// TwinCAT 3 PLC project Main
// ProgramVersion: 3.1.4026.10
// libraries:
//   Tc2_EtherCAT, * (Beckhoff Automation GmbH)
//   Tc2_IoFunctions, * (Beckhoff Automation GmbH)
//   Tc2_Math, * (Beckhoff Automation GmbH)
//   Tc2_MC2, * (Beckhoff Automation GmbH)
//   Tc2_NC, * (Beckhoff Automation GmbH)
//   Tc2_Standard, * (Beckhoff Automation GmbH)
//   Tc2_System, * (Beckhoff Automation GmbH)
//   Tc2_Utilities, * (Beckhoff Automation GmbH)
//   Tc3_EventLogger, * (Beckhoff Automation GmbH)
//   Tc3_McCollisionAvoidance, * (Beckhoff Automation GmbH)
//   Tc3_McCoordinatedMotion, * (Beckhoff Automation GmbH)
//   Tc3_Module, * (Beckhoff Automation GmbH)
//   Tc3_XTS_Utility, * (Beckhoff Automation GmbH)
// project tree:
//   DUTs/delete/ MainCommands_typ.TcDUT, MainStateMachine_enum.TcDUT (not stored), MainState_enum.TcDUT, MediatorGroupStatus.TcDUT (not stored), MotionParameters_typ.TcDUT (not stored), MoverCommandType_enum.TcDUT (not stored), MoverState_enum.TcDUT (not stored), PositionTriggerStats_typ.TcDUT (not stored), StationStats_typ.TcDUT (not stored), TrackCyclicState.TcDUT (not stored), TrackInfo.TcDUT (not stored), TrackState.TcDUT (not stored), UserStationsMonitor.TcDUT (not stored)
//   DUTs/ M1Detection.TcDUT (not stored), MoverControlFlags.TcDUT, MoverSequence.TcDUT, StationSequence.TcDUT (not stored), XTSSequence.TcTLEO
//   / GlobalTextList.TcGTLO (not stored), PlcTask.TcTTO
//   GVLs/ GVL.TcGVL, HMI.TcGVL, IOGVL.TcGVL, SafetyGVL.TcGVL
//   ITFs/ iMoverList.TcIO (not stored), iMover.TcIO, iTrack.TcIO (not stored)
//   POUs/ Main.TcPOU
//   POUs/XTS/ Mover.TcPOU, Station.TcPOU, Zone.TcPOU

CONFIGURATION Main
    RESOURCE PLC ON TwinCAT3
        TASK PlcTask(INTERVAL := T#1ms, PRIORITY := 6);
        PROGRAM Main WITH PlcTask : Main;
    END_RESOURCE
END_CONFIGURATION

// ---- DUTs/delete/MainCommands_typ.TcDUT
TYPE MainCommands_typ :
    STRUCT

        Enable  : BOOL; // Enables Movers & Collision Avoidance, activates M1 Detection
        Start   : BOOL; // Issues initial command, starts motion
        Stop    : BOOL; // Stops movers, deregisters movers from all objectives	
        Disable : BOOL; // Disables Movers, Ungroups Movers

    END_STRUCT
END_TYPE

// ---- DUTs/delete/MainState_enum.TcDUT
{attribute 'strict'}
{attribute 'to_string'}
TYPE MainState_enum : (
        MS_DISABLED					:= 0,
		MS_INITIALIZING_XPU			:= 5,
        MS_INITIALIZING_MOVERS		:= 10,
		MS_ONESHOT_ENABLE			:= 20,
        MS_ENABLING_MOVERS			:= 30,
        MS_INITIALIZING_OBJECTIVES	:= 40,
		MS_INITIALIZE_TRACKS		:= 44,
		MS_ACTIVATE_TRACKS			:= 45,
		MS_WAIT_FOR_TRACKS			:= 46,
        MS_ENABLED					:= 50,
        MS_RUN						:= 60,
		MS_ONESHOT_STOP				:= 70,
        MS_STOPPING					:= 80,
        MS_STOPPED					:= 90,
		MS_ONESHOT_DISABLE			:= 100,
        MS_DISABLING				:= 110,
        MS_ERROR					:= 120,
        MS_DEBUG					:= 1000
    );
END_TYPE

// ---- DUTs/MoverControlFlags.TcDUT
TYPE MoverControlFlags :
STRUCT

	loadTray_Busy		: BOOL;			// To the machine to check Sensor
	loadTray_Complete	: BOOL;			// From Sensor is TRUE
	loadArea1_Busy		: BOOL;			// TO Robot 1 to start working
	loadArea1_Complete	: BOOL;			// FROM Robot 1 that placing parts has completed
	loadArea2_Busy		: BOOL;			// TO Robot 2 to start working
	loadArea2_Complete	: BOOL;			// FROM Robot 1 that placing parts has completed
	loadArea3_Busy		: BOOL;			// TO Robot 3 to start working
	loadArea3_Complete	: BOOL;			// FROM Robot 1 that placing parts has completed
	loadArea4_Busy		: BOOL;			// TO Robot 4 to start working
	loadArea4_Complete	: BOOL;			// From Robot 1 that placing parts has completed
	unloadTray_Busy		: BOOL;			// To Robot 5 to start working
	unloadTray_Complete	: BOOL;			// From Robot 5. Tray is unloaded



END_STRUCT
END_TYPE

// ---- DUTs/MoverSequence.TcDUT
{attribute 'qualified_only'}
{attribute 'strict'}
TYPE MoverSequence :
(
	Off,
	Idle,
	MovingToStart,
	AtStart,
	MovingToStation,
	AtStation,
	MovingToQueue,
	AtQueue,
	Error,
	Stop,
	Stopping,
	RemoveAxes,
	RemovingAxes,
	Pausing,
	Paused,
	Disabling,
	Disabled,
	Reset,
	Resetting,
	Waiting	
);
END_TYPE

// ---- DUTs/XTSSequence.TcTLEO
{attribute 'qualified_only'}
{attribute 'strict'}
TYPE XTSSequence :
(
	Off,
	EnableMovers,
	EnableGroup,
	AddAxes,
	RemoveAxes,
	RemovedAxes,
	DisableMovers,
	Disabled,
	Start,
	Run,
	Stop,
	Stopping,
	Paused,
	Standby,
	Error,
	Waiting
);
END_TYPE

// ---- GVLs/GVL.TcGVL
{attribute 'qualified_only'}
VAR_GLOBAL CONSTANT

    pXtsProcessingUnit : OTCID	:=	01010090;	 

	TRACK_LENGTH 				: LREAL := 7000; // This should be set to the exact length [mm] of the track system
	NUM_MOVERS   				: USINT := 20;   // This should be set to the exact number of movers on the system
	
	// The following should be set to a value **equal to or greater than** the number of objectives needed
	NUM_POSITIONTRIGGERS		: USINT := 10;	// Position Triggers
	NUM_STATIONS				: USINT := 8;	// Stations
	NUM_ZONES					: USINT := 10;	// Zones

	// Station constants
	startStation				: USINT	:= 1;		// set this number to the index of the station all movers should start from
	stationTolerance			: LREAL	:= 0.5;		// set to number of millimeters tolerance for mover at station
	zeroSpeed					: LREAL	:= 10.0;		// tolerance for definition of not moving

END_VAR
VAR_GLOBAL
	Mover			: ARRAY[1..GVL.NUM_MOVERS] OF Mover;
	Station			: ARRAY[1..GVL.NUM_STATIONS] OF station;
	Zone			: ARRAY[1..GVL.NUM_ZONES] OF zone;
	newCallTime: LREAL;
	
	//-------------ADDED BY NIJAZ-------------
	dsMoverControlFlags		:	MoverControlFlags;
	
END_VAR

// ---- GVLs/HMI.TcGVL
{attribute 'qualified_only'}
VAR_GLOBAL
	Start					: BOOL;
	E_Stop					: BOOL;
	Stop					: BOOL;
	Resume					: BOOL;
	ResetXTS_Error			: BOOL;
	bzone0Stop				: BOOL;
	SafeToUnlock			: BOOL;
	dsMoverControlFlags		: MoverControlFlags;
	ShuttleMover			: BOOL;
	
	
	//Linked to SAFETY Alias
	LockDoors		AT %Q*	: BOOL;		
	
END_VAR

// ---- GVLs/IOGVL.TcGVL
{attribute 'qualified_only'}
VAR_GLOBAL
	
//INPUTS
iTrayDetectSensor	AT %I*	:	BOOL;
iDoor1Opened		AT %I*	:	BOOL;		
iDoor2Opened		AT %I*	:	BOOL;
iDoor3Opened		AT %I*	:	BOOL;
iDoor4Opened		AT %I*	:	BOOL;
iMainAirPressure 	AT %I*	:	BOOL;

//------XTS Power Monitor Breakers	
//- EL1809 Mod1
iCircuitBreaker24VDC			AT %I*	:	BOOL;
iCircuitBreakerSafety			AT %I*	:	BOOL;
iXTS_Module1					AT %I*	:	BOOL;
iXTS_Module2					AT %I*	:	BOOL;
iXTS_Module3					AT %I*	:	BOOL;
iXTS_Module4					AT %I*	:	BOOL;
iXTS_Module5					AT %I*	:	BOOL;
iXTS_Module6					AT %I*	:	BOOL;
iLubricationOn					AT %I*	:	BOOL;
//- EL1809 Mod2
iPowerSupply48VDC1				AT %I*	:	BOOL;
iPowerSupply48VDC2				AT %I*	:	BOOL;
iPowerSupply48VDC3				AT %I*	:	BOOL;
iLubricationLevelOK				AT %I*	:	BOOL;
iLubricationDone				AT %I*	:	BOOL;
iCircuitBreaker48VDC1			AT %I*	:	BOOL;
iCircuitBreaker48VDC2			AT %I*	:	BOOL;
iCircuitBreaker48VDC3			AT %I*	:	BOOL;
iCircuitBreakerXTSModule1		AT %I*	:	BOOL;
iCircuitBreakerXTSModule2		AT %I*	:	BOOL;
iCircuitBreakerXTSModule3		AT %I*	:	BOOL;
iCircuitBreakerXTSModule4		AT %I*	:	BOOL;
iCircuitBreakerXTSModule5		AT %I*	:	BOOL;
iCircuitBreakerXTSModule6		AT %I*	:	BOOL;
iBrakeResistorON				AT %I*	:	BOOL;

//-----------------------------------------------------------------------------------------------------------------------------------
//OUTPUTS
oBacklight1			AT %Q*	:	BOOL;
oBacklight2			AT %Q*	:	BOOL;
oBacklight3			AT %Q*	:	BOOL;
oBacklight4			AT %Q*	:	BOOL;
oBacklight5			AT %Q*	:	BOOL;
oBacklight6			AT %Q*	:	BOOL;
oBacklight7			AT %Q*	:	BOOL;
oBacklight8			AT %Q*	:	BOOL;
oBacklight9			AT %Q*	:	BOOL;
oBacklight10		AT %Q*	:	BOOL;
oBacklight11		AT %Q*	:	BOOL;
oBacklight12		AT %Q*	:	BOOL;
oBacklight13		AT %Q*	:	BOOL;
oBacklight14		AT %Q*	:	BOOL;
oBacklight15		AT %Q*	:	BOOL;
oBacklight16		AT %Q*	:	BOOL;
oEStopLight			AT %Q*	:	BOOL;
oConveyor			AT %Q*	:	BOOL;
oLubeON				AT %Q*	:	BOOL;


END_VAR

// ---- GVLs/SafetyGVL.TcGVL
{attribute 'qualified_only'}
VAR_GLOBAL
	
//OUTPUTS TO SAFETY GROUP
err_ack			AT %Q*	:	BOOL;
run				AT %Q*	:	BOOL := TRUE;
DoorsClosed 	AT %Q*	:	BOOL;
ResetCurtains	AT %Q*	:	BOOL;

//INPUTS FROM SAFETY GROUP
CurtainsOK		AT %I*	:	BOOL;
AllSafetyOK		AT %I*	:	BOOL;
EStopStatus		AT %I*	:	BOOL;

END_VAR

// ---- ITFs/iMover.TcIO
INTERFACE iMover

METHOD ActivateTrack : BOOL
VAR_INPUT
	Track	: REFERENCE TO Track;
END_VAR
END_METHOD

{attribute 'monitoring' := 'call'}
PROPERTY CurrentDestinationPosition : LREAL
GET
END_GET
END_PROPERTY

PROPERTY CurrentDestinationTrack : DINT
GET
END_GET
END_PROPERTY

{attribute 'monitoring' := 'call'}
PROPERTY CurrentMoveType : MoverCommandType_enum
GET
END_GET
END_PROPERTY

PROPERTY CurrentObjective : String
GET
END_GET
END_PROPERTY

PROPERTY CurrentTrack : POINTER TO Track
GET
END_GET
END_PROPERTY

METHOD Cyclic : iMover
VAR_IN_OUT
	GroupReference		: AXES_GROUP_REF;
END_VAR
END_METHOD

METHOD Disable : iMover
VAR_INPUT
END_VAR
END_METHOD

METHOD Enable : iMover
VAR_INPUT
END_VAR
END_METHOD

METHOD GroupStop : iMover
VAR_INPUT
END_VAR
END_METHOD

METHOD Halt : iMover
VAR_INPUT
END_VAR
END_METHOD

PROPERTY IsTrackReady : BOOL
GET
END_GET
END_PROPERTY

METHOD LogUserEvent : iMover
VAR_INPUT
	String1	: STRING;	// First content section of user-event message
	String2 : STRING;	// Second content section of user-event message
	String3 : STRING;	// Third content section of user-event message
END_VAR
END_METHOD

METHOD PUBLIC MoveToPosition : iMover
VAR_INPUT
	
	DestinationPosition		: LREAL;	// position on track for a shuttle to move towards

END_VAR
END_METHOD

METHOD MoveToStation : iMover
VAR_INPUT
	DestinationStation	: REFERENCE TO delete_Station;	
END_VAR
END_METHOD

METHOD MoveVelocity : iMover
VAR_INPUT
	DesiredVelocity : LREAL;		//The velocity to be commanded [mm/s]
END_VAR
END_METHOD

PROPERTY Payload : USINT
GET
END_GET
SET
END_SET
END_PROPERTY

METHOD ReissueCommand : iMover
VAR_INPUT
END_VAR
END_METHOD


METHOD SetAcceleration : iMover
VAR_INPUT
	Acceleration	: LREAL;
END_VAR
END_METHOD

METHOD SetDeceleration : iMover
VAR_INPUT
	Deceleration	: LREAL;
END_VAR
END_METHOD

METHOD SetDirection : iMover
VAR_INPUT
	Direction		: Tc3_Mc3Definitions.MC_Direction;
END_VAR
END_METHOD

METHOD SetGap : iMover
VAR_INPUT
	Gap	: LREAL;
END_VAR
END_METHOD

METHOD SetGapMode : iMover
VAR_INPUT
	Mode	: MC_GAP_CONTROL_MODE;
END_VAR
END_METHOD

METHOD SetJerk : iMover
VAR_INPUT
	Jerk		: LREAL;
END_VAR
END_METHOD

METHOD SetVelocity : iMover
VAR_INPUT
	Velocity		: LREAL;		// Updates Mover's internal velocity parameter. Takes effect immediately. [mm/s]
END_VAR
END_METHOD

METHOD SyncToAxis : iMover
VAR_INPUT
	
	MasterAxis		: REFERENCE TO AXIS_REF;
	MasterSyncPos	: LREAL;	// Master sync position (nonmodulo), where the input axis will be located when first synchronized
	SlaveSyncPos	: LREAL;	// Mover sync position, where the mover will be located when first synchronized
	SyncStrategy	: MC_SYNC_STRATEGY;	// Direction input
	
END_VAR
END_METHOD

METHOD SyncToMover : iMover
VAR_INPUT

	MasterMover		: REFERENCE TO delete_Mover;	// Synchronization master mover, whose position to follow. Further motion commands break the pairing
	Gap				: LREAL;				// Gap distance to lead mover. Positive values indicate following, negative values indicate leading

END_VAR
END_METHOD

END_INTERFACE

// ---- POUs/Main.TcPOU
PROGRAM Main
VAR
	PowerOn					: BOOL	:= TRUE;	// initialize on, turn false on second scan
	FirstRun				: BOOL := TRUE;		// initialize on, turn false when system has reached starting postion 
	i						: UINT;								// loop index variable
	Step					: XTSSequence;						// primary sequencer
	stCaGroupRef			: AXES_GROUP_REF;
	fbEnableGroup			: MC_GroupEnable;
	fbAddAxis				: ARRAY[1..GVL.NUM_MOVERS] OF MC_AddAxisToGroup;
	fbRemoveAxisFromGroup	: ARRAY[1..GVL.NUM_MOVERS] OF MC_RemoveAxisFromGroup;
	nAtStart				: UINT;
	nToStart				: UINT;
	allMoversHalted			: BOOL;	
	MoversReady				: BOOL;
	Started					: BOOL;		
	Resumed					: BOOL;
	bLightCurtainExited		: R_TRIG;
	bLightCurtainEntered	: F_TRIG;
	bEstopPressed			: F_TRIG;
	safeToOpenDoors			: BOOL;
	allMoversNotMoving		: BOOL;
	DelayMoversTimer		: TON;
	
	//Timers for generating a pulse
	PulseTON	: TON;
	PulseTOF	: TOF;
	OnDuration	: TIME := T#500MS;
	OFFDuration	: TIME := T#1000MS;
	bCycleBit	: BOOL;
	
	//M1 Detection
	fbReadM1DetectMode		: ADSREAD;
	fbReadM1DetectValid		: ADSREAD;
	fbReadM1DetectActive	: ADSREAD;
	fbWriteM1Detect			: ADSWRITE;
	fbDelayM1Timer			: TON;
	IsIdDetectionActive		: BOOL;			// M1 Detection currently underway
	Mover1Found				: BOOL;			// M1 Detection has completed
	Mover1Error				: BOOL;			// M1 Detection has Failed
	M1DetectStep			: M1Detection;	
	M1DetectAttemptCounter	: INT;
END_VAR

(* this program handles the main sequencer of this machine *)

// cyclic call to execute fb's for movers, stations, and zones
FOR i := 1 TO GVL.NUM_MOVERS DO
	GVL.Mover[i]();
	GVL.Mover[i].AxisReference.ReadStatus();
	fbRemoveAxisFromGroup[i](AxesGroup		:= stCaGroupRef);
	fbAddAxis[i](AxesGroup		:= stCaGroupRef,
				Axis			:= GVL.Mover[i].AxisReference);
	//Monitoring if all movers are in stopped motion state			
	IF GVL.Mover[i].AxisReference.Status.Moving THEN
		allMoversNotMoving	:= FALSE;
	ELSE
		allMoversNotMoving	:= TRUE;
	END_IF
	
END_FOR
FOR i := 1 TO GVL.NUM_STATIONS DO
	GVL.Station[i]();
END_FOR
FOR i := 1 TO gvl.NUM_ZONES DO
	GVL.Zone[i]();
END_FOR

IF HMI.ResetXTS_Error THEN
	FOR i := 1 TO GVL.NUM_MOVERS DO
		GVL.Mover[i].toReset := TRUE;
	END_FOR
	HMI.ResetXTS_Error := FALSE;
END_IF


// check for E-STOP
bEstopPressed(CLK:=SafetyGVL.EStopStatus);
IF bEstopPressed.Q OR HMI.E_Stop THEN
	Step			:= XTSSequence.Stop;
	HMI.E_Stop := FALSE;
END_IF

CASE Step OF

//-----------------------------------------------------------------------------------------------------------------------	
	XTSSequence.Off:
		IF SafetyGVL.EStopStatus AND IOGVL.iPowerSupply48VDC1 AND IOGVL.iPowerSupply48VDC2 AND IOGVL.iPowerSupply48VDC3 AND Mover1Found = FALSE THEN
			Initialize();
		END_IF
		// state waiting for HMI.Start
		IF HMI.Start AND Mover1Found THEN
			Step		:= XTSSequence.EnableMovers;
			Started 	:= TRUE;
			HMI.Start 	:= FALSE;
		END_IF

//-----------------------------------------------------------------------------------------------------------------------	
	XTSSequence.Paused:
		//state waiting for HMI.Start or HMI.Resume
		IF HMI.Start THEN
			Step		:= XTSSequence.EnableMovers;
			Started 	:= TRUE;
			HMI.Start 	:= FALSE;
		END_IF
	
		IF HMI.Resume THEN
			Step		:= XTSSequence.EnableMovers;
			Resumed 	:= TRUE;
			HMI.Resume 	:= FALSE;
			HMI.Stop  	:= FALSE;
		END_IF
	
//-----------------------------------------------------------------------------------------------------------------------	
	XTSSequence.Stop:
	
	FOR i := 1 TO GVL.NUM_MOVERS  DO
		GVL.Mover[i].toStop := TRUE;
	END_FOR
	
	Started 	:= FALSE;
	Resumed 	:= FALSE;
	Step		:= XTSSequence.Stopping;
		
//-----------------------------------------------------------------------------------------------------------------------	
	XTSSequence.Stopping:
		// Waiting for all to come to a full stop
		
	allMoversHalted		:= TRUE;
	
		FOR i := 1 TO GVL.NUM_MOVERS DO
			IF GVL.Mover[i].AxisReference.Status.Moving THEN
				allMoversHalted		:= FALSE;
			END_IF
		END_FOR
	
	IF allMoversHalted THEN
		Step		:= XTSSequence.RemoveAxes;
	END_IF
	
//-----------------------------------------------------------------------------------------------------------------------	
	XTSSequence.RemoveAxes:
		// remove all axes to collision avoidance group
		// loop through each mover axis and remove CA group
		FOR i:= 1 TO GVL.NUM_MOVERS DO
			fbRemoveAxisFromGroup[i].IdentInGroup := UDINT_TO_IDENTINGROUP(UINT_TO_UDINT(i));
			fbRemoveAxisFromGroup[i].Execute			:= TRUE;
		END_FOR
	
		IF stCaGroupRef.NcToPlc.CA.Common.GroupAxesCount = 0 THEN
			FOR i:= 1 TO GVL.NUM_MOVERS DO
				fbRemoveAxisFromGroup[i].IdentInGroup	:= UDINT_TO_IDENTINGROUP(UINT_TO_UDINT(i));
				fbRemoveAxisFromGroup[i].Execute			:= FALSE;
				MoversReady := FALSE;
		END_FOR
			Mover1Found := FALSE;
			Step := XTSSequence.DisableMovers;
		END_IF

//-----------------------------------------------------------------------------------------------------------------------	
	XTSSequence.DisableMovers:
	FOR i := 1 TO GVL.NUM_MOVERS  DO
		GVL.Mover[i].toDisable := TRUE;
	END_FOR
	
	Step := XTSSequence.Off;
		
//-----------------------------------------------------------------------------------------------------------------------			
	XTSSequence.EnableMovers:
		// enable all movers
		FOR i := 1 TO GVL.NUM_MOVERS DO
			IF NOT GVL.Mover[i].Enabled THEN
				GVL.Mover[i].Enable	:= TRUE;
			END_IF
		END_FOR
		
		// check for all enabled
		FOR i := 1 TO GVL.NUM_MOVERS DO
			IF NOT GVL.Mover[i].Enabled THEN
				// not enabled, leave for loop
				EXIT;
			END_IF
			// made it this far, all movers are enabled
			IF i = gvl.NUM_MOVERS THEN
				Step	:= XTSSequence.EnableGroup;
			END_IF
		END_FOR
		
//-----------------------------------------------------------------------------------------------------------------------		
	XTSSequence.EnableGroup:
	// enable CA group
	fbEnableGroup.Execute := TRUE;
	// verify group enabled successfully
	IF fbEnableGroup.Done = TRUE THEN
		fbEnableGroup.Execute := FALSE;
		Step := XTSSequence.AddAxes;
	END_IF
		
//-----------------------------------------------------------------------------------------------------------------------		
	XTSSequence.AddAxes:
		// add all axes to collision avoidance group
		// loop through each mover axis and add to CA group
	FOR i:= 1 TO GVL.NUM_MOVERS DO
		fbAddAxis[i].IdentInGroup := UDINT_TO_IDENTINGROUP(UINT_TO_UDINT(i));
		fbAddAxis[i].Execute := TRUE;
	END_FOR
	
	// verify all axes added
	IF stCaGroupRef.NcToPlc.CA.Common.GroupAxesCount = GVL.NUM_MOVERS THEN
		FOR i:= 1 TO GVL.NUM_MOVERS DO
			fbAddAxis[i].IdentInGroup := UDINT_TO_IDENTINGROUP(UINT_TO_UDINT(i));
			fbAddAxis[i].Execute := FALSE;
			Step	:= XTSSequence.StandBy;
		END_FOR
	END_IF
		
//-----------------------------------------------------------------------------------------------------------------------		
	XTSSequence.StandBy:
	IF Started THEN
		// first time code executes this far (after power on) move to a start position
		Started := FALSE;
		Step	:= XTSSequence.Start;
	ELSIF Resumed THEN
		// any other time code executes here, resume operation where movers left off
		Resumed := FALSE;
		Step	:= XTSSequence.Run;
	END_IF

//-----------------------------------------------------------------------------------------------------------------------		
	XTSSequence.Start:
		// request all movers proceed to starting station
IF HMI.bzone0Stop = FALSE THEN
	FOR i:= 1 TO GVL.NUM_MOVERS DO
		GVL.Mover[i].toStart	:= TRUE;
	END_FOR
	// verify one mover is at start, all others have commands and are at zero speed
	nAtStart	:= 0;
	nToStart	:= 0;
	FOR i:= 1 TO GVL.NUM_MOVERS DO
		IF GVL.Mover[i].Step = MoverSequence.AtStart THEN
			nAtStart	:= nAtStart + 1;
		ELSIF GVL.Mover[i].Step = MoverSequence.MovingToStart THEN
			nToStart	:= nToStart + 1;
		END_IF
	END_FOR
	IF nAtStart = 1 AND nToStart = GVL.NUM_MOVERS - 1 THEN
		Step	:= XTSSequence.Run;
	END_IF
END_IF	
//-----------------------------------------------------------------------------------------------------------------------	
	XTSSequence.Run:

IF HMI.Stop = FALSE THEN
	
	// LOAD TRAY STATION
	IF GVL.Station[1].Step = StationSequence.MoverPresent THEN
		HMI.dsMoverControlFlags.loadTray_Busy := TRUE;
		IF HMI.dsMoverControlFlags.loadTray_Complete THEN			//IF SENSOR IS TRUE PACKAGE IS PRESENT MOVER GOES TO NEXT STATION
			HMI.dsMoverControlFlags.loadTray_Complete := FALSE;
			GVL.Station[1].bMoveToNext := TRUE;
		END_IF
	ELSE
		HMI.dsMoverControlFlags.loadTray_Busy := FALSE;
	END_IF
	
	// INSPECT TRAY STATION
	IF GVL.Station[2].Step = StationSequence.MoverPresent THEN
		HMI.dsMoverControlFlags.inspectTray_Busy := TRUE;
		IF HMI.dsMoverControlFlags.inspectTray_Complate THEN			//IF SENSOR IS TRUE PACKAGE IS PRESENT MOVER GOES TO NEXT STATION
			HMI.dsMoverControlFlags.inspectTray_Complate := FALSE;
			GVL.Station[2].bMoveToNext := TRUE;
		END_IF
	ELSE
		HMI.dsMoverControlFlags.inspectTray_Busy := FALSE;
	END_IF
	
	// LOAD PARTS STATION 1
	IF GVL.Station[3].Step = StationSequence.MoverPresent THEN
		HMI.dsMoverControlFlags.loadArea1_Busy := TRUE;				//SIGNAL TO ROBOT 1 TO LOAD PARTS
		IF HMI.dsMoverControlFlags.loadArea1_Complete THEN			//SIGNAL FROM ROBOT 1 PARTS COMPLETED
			HMI.dsMoverControlFlags.loadArea1_Complete := FALSE;
			GVL.Station[3].bMoveToNext := TRUE;
		END_IF
	ELSE 
		HMI.dsMoverControlFlags.loadArea1_Busy := FALSE;
	END_IF
	
	// LOAD PARTS STATION 2
	IF GVL.Station[4].Step = StationSequence.MoverPresent THEN
		HMI.dsMoverControlFlags.loadArea2_Busy := TRUE;				//SIGNAL TO ROBOT 2 TO LOAD PARTS
		IF HMI.dsMoverControlFlags.loadArea2_Complete THEN			//SIGNAL FROM ROBOT 2 PARTS COMPLETED
			HMI.dsMoverControlFlags.loadArea2_Complete := FALSE;
			GVL.Station[4].bMoveToNext := TRUE;
		END_IF
	ELSE
		HMI.dsMoverControlFlags.loadArea2_Busy := FALSE;	
	END_IF
	
	// LOAD PARTS STATION 3
	IF GVL.Station[5].Step = StationSequence.MoverPresent THEN
		HMI.dsMoverControlFlags.loadArea3_Busy := TRUE;				//SIGNAL TO ROBOT 3 TO LOAD PARTS
		IF HMI.dsMoverControlFlags.loadArea3_Complete THEN			//SIGNAL FROM ROBOT 3 PARTS COMPLETED
			HMI.dsMoverControlFlags.loadArea3_Complete := FALSE;
			GVL.Station[5].bMoveToNext := TRUE;
		END_IF
	ELSE
		HMI.dsMoverControlFlags.loadArea3_Busy := FALSE;
	END_IF

	// LOAD PARTS STATION 4
	IF GVL.Station[6].Step = StationSequence.MoverPresent THEN
		HMI.dsMoverControlFlags.loadArea4_Busy := TRUE;				//SIGNAL TO ROBOT 4 TO LOAD PARTS
		IF HMI.dsMoverControlFlags.loadArea4_Complete THEN			//SIGNAL FROM ROBOT 4 PARTS COMPLETED
			HMI.dsMoverControlFlags.loadArea4_Complete := FALSE;
			GVL.Station[6].bMoveToNext := TRUE;
		END_IF
	ELSE
		HMI.dsMoverControlFlags.loadArea4_Busy := FALSE;	
	END_IF
	
	// UNLOAD PARTS STATION 
	IF GVL.Station[7].Step = StationSequence.MoverPresent THEN
		HMI.dsMoverControlFlags.unloadTray_Busy := TRUE;			//SIGNAL TO ROBOT 5 TO UNLOAD TRAY
		IF HMI.dsMoverControlFlags.unloadTray_Complete THEN			//SIGNAL FROM ROBOT 5 UNLOAD TRAY COMPLETED
			HMI.dsMoverControlFlags.unloadTray_Complete := FALSE;
			IF HMI.bzone0Stop THEN
				GVL.Station[7].bMoveToNext := TRUE;					//Send to Queue Movers Station
			ELSE
				GVL.Station[7].bMoveToStart := TRUE;				//Send to Load Tray Station
			END_IF

		END_IF
	ELSE
		HMI.dsMoverControlFlags.unloadTray_Busy := FALSE;
	END_IF
	
	// Queue Station used only if Operator is in Zone 1
	IF GVL.Station[8].Step = StationSequence.MoverPresent THEN
		IF HMI.bzone0Stop = FALSE THEN			
			GVL.Station[8].bMoveToStart := TRUE;
		END_IF
	END_IF
	
	
	// Starting over on the condition that movers are stationary and HMI.Startover has been pressed.
	IF allMoversNotMoving THEN				
		IF HMI.Start THEN
			FOR i := 2 TO GVL.NUM_STATIONS DO
				IF GVL.Station[i].Step = StationSequence.MoverPresent THEN
				GVL.Station[i].bMoveToStart := TRUE;
				END_IF
			END_FOR	
			HMI.Start := FALSE;
		END_IF
	END_IF
	
ELSE
	
	Step	:= XTSSequence.Paused;
	
END_IF

END_CASE

fbEnableGroup(AxesGroup	:= stCaGroupRef);
LightCurtainCheck();
ShuttleMoverToQueue();
DoorsClosedMonitor();


IF allMoversNotMoving THEN
	HMI.SafeToUnlock := TRUE;
ELSE
	HMI.SafeToUnlock := FALSE;
END_IF

ACTION DoorsClosedMonitor:





IF IOGVL.iDoor1Opened OR IOGVL.iDoor2Opened OR IOGVL.iDoor3Opened OR IOGVL.iDoor4Opened THEN
	SafetyGVL.DoorsClosed := FALSE;
ELSE
	SafetyGVL.DoorsClosed := TRUE;
END_IF


PulseTON(IN := NOT SafetyGVL.AllSafetyOK AND NOT bCycleBit, PT := OnDuration);
PulseTOF(IN := bCycleBit, PT := OFFDuration);

IF PulseTON.Q THEN
	bCycleBit := TRUE;
	IOGVL.oEStopLight := TRUE;
ELSE 
	IOGVL.oEStopLight := FALSE;
END_IF

IF PulseTOF.Q THEN
	bCycleBit := FALSE;
END_IF
END_ACTION

METHOD Initialize : BOOL
VAR_INPUT
END_VAR
// set values of function blocks
	GVL.Station[1].Position		:= 0.0;				//	Load Tray
	GVL.Station[2].Position		:= 750.0;			//	Inspect Tray
	GVL.Station[3].Position		:= 1500.0;			//	Load Parts 1
	GVL.Station[4].Position		:= 2250.0;			//	Load Parts 2
	GVL.Station[5].Position		:= 3000.0;			//	Load Parts 3
	GVL.Station[6].Position		:= 3600.0;			//	Load Parts 4
	GVL.Station[7].Position		:= 4250.0;			//	Unload Tray
	GVL.Station[8].Position		:= 4449.0;			//	Queue Area if operator is in workspace
	
	CASE M1DetectStep OF		//This Case statement will make 10 attempts to find Mover1 and error if not successful
		
M1Detection.Read:// ------------------------------------------------------- Determine current M1 Detection Status
		
	fbWriteM1Detect.WRITE			:= FALSE;
	
	fbReadM1DetectValid.NETID		:= '';
	fbReadM1DetectValid.PORT		:= 351;
	fbReadM1DetectValid.IDXGRP		:= GVL.pXtsProcessingUnit;
	fbReadM1DetectValid.IDXOFFS		:= 16#03080251;
	fbReadM1DetectValid.LEN			:= SIZEOF( Mover1Found );
	fbReadM1DetectValid.DESTADDR	:= ADR( Mover1Found );
	fbReadM1DetectValid.READ		:= TRUE;
	
	fbReadM1DetectActive.NETID		:= '';
	fbReadM1DetectActive.PORT		:= 351;
	fbReadM1DetectActive.IDXGRP		:= GVL.pXtsProcessingUnit;
	fbReadM1DetectActive.IDXOFFS	:= 16#03080268;
	fbReadM1DetectActive.LEN		:= SIZEOF( IsIdDetectionActive );
	fbReadM1DetectActive.DESTADDR	:= ADR( IsIdDetectionActive );
	fbReadM1DetectActive.READ		:= TRUE;
	
	M1DetectStep 					:= M1Detection.ReadBuffer;
		
M1Detection.ReadBuffer:// ------------------------------------------------------- Buffer

	fbDelayM1Timer( IN := TRUE, PT := T#3000MS );
	IF fbDelayM1Timer.Q THEN
		fbDelayM1Timer.IN				:= FALSE;
		fbReadM1DetectValid.READ		:= FALSE;
		fbReadM1DetectActive.READ		:= FALSE;
		M1DetectAttemptCounter := M1DetectAttemptCounter + 1;
		M1DetectStep 			:= M1Detection.Analyze;
	END_IF
		
M1Detection.Analyze:// ------------------------------------------------------- Determine to activate M1 Detect or ignore
	
IF M1DetectAttemptCounter < 10 THEN
	IF IsIdDetectionActive THEN
		M1DetectStep					:= M1Detection.Read;
	ELSIF Mover1Found THEN
		M1DetectStep					:= M1Detection.Done;	// M1 Detection complete, ready to enable this mover
	ELSE
		M1DetectStep					:= M1Detection.Write;	// M1 Detection hasn't been started yet. So start it!	
	END_IF
ELSE
	M1DetectStep				:= M1Detection.Error;	// M1 Detection Failed
END_IF

M1Detection.Write:// ------------------------------------------------------- Begin M1 Detection

	fbWriteM1Detect.NETID			:= '';
	fbWriteM1Detect.PORT			:= 351;
	fbWriteM1Detect.IDXGRP			:= GVL.pXtsProcessingUnit;
	fbWriteM1Detect.IDXOFFS			:= 16#03080250;
	fbWriteM1Detect.WRITE			:= TRUE;

	M1DetectStep 					:= M1Detection.WriteBuffer;
		
M1Detection.WriteBuffer:// ------------------------------------------------------- Buffer

	fbDelayM1Timer( IN := TRUE, PT := T#2000MS );
		
	IF fbDelayM1Timer.Q THEN
		fbDelayM1Timer.IN				:= FALSE;
		fbWriteM1Detect.WRITE			:= FALSE;
		M1DetectStep 					:= M1Detection.Read;
	END_IF

M1Detection.Done:// ------------------------------------------------------- Finished M1 Detection

	Mover1Found := TRUE;
	IsIdDetectionActive := FALSE;
	M1DetectStep 					:= M1Detection.Read;

M1Detection.Error:// ------------------------------------------------------- Failed M1 Detection

	Mover1Error			:= TRUE;
	IsIdDetectionActive := FALSE;

END_CASE

fbReadM1DetectValid();
fbReadM1DetectActive();
fbWriteM1Detect();
fbDelayM1Timer();
END_METHOD

ACTION LightCurtainCheck:
// ZONE 0  OPERATER LOADING
(*
IF SafetyGVL.AllSafetyOK THEN
	bLightCurtainEntered(CLK:=SafetyGVL.CurtainsOK);
	bLightCurtainExited(CLK:=SafetyGVL.CurtainsOK);
		IF bLightCurtainEntered.Q THEN
			FOR i:= 1 TO GVL.NUM_MOVERS DO	
				IF GVL.Mover[i].Position > 4500.0 THEN
				GVL.Mover[i].toPause	:= TRUE;
				GVL.Mover[i].toNext		:= FALSE;
				GVL.Mover[i].toStart	:= FALSE;
				END_IF
			END_FOR
		END_IF
		
		IF bLightCurtainExited.Q THEN
			DelayMoversTimer( IN := TRUE, PT := T#1000MS );
		ELSIF bLightCurtainEntered.Q THEN
			DelayMoversTimer.IN := FALSE;
		END_IF
		
		IF DelayMoversTimer.Q THEN
			FOR i:= 1 TO GVL.NUM_MOVERS DO	
				IF GVL.Mover[i].Position > 4500.0 THEN
					GVL.Mover[i].toStart	:= TRUE;
				END_IF
			END_FOR
		END_IF
END_IF
	*)
END_ACTION

ACTION ShuttleMoverToQueue:

// This will be used for set up if mover is needed to be re-circulated around track

IF 	GVL.Station[1].Step = StationSequence.MoverPresent AND 
	GVL.Station[2].Step = StationSequence.Idle AND 
	GVL.Station[3].Step = StationSequence.Idle AND 
	GVL.Station[4].Step = StationSequence.Idle AND 
	GVL.Station[5].Step = StationSequence.Idle AND 
	GVL.Station[6].Step = StationSequence.Idle AND 
	GVL.Station[7].Step = StationSequence.Idle AND 
	HMI.ShuttleMover THEN
		GVL.Station[1].bMoveToQueue := TRUE;
		HMI.ShuttleMover := FALSE;
		
	(*FOR i:= 1 TO GVL.NUM_STATIONS DO
		GVL.Station[i].
	END_FOR
	*)
END_IF
END_ACTION

END_PROGRAM

// ---- POUs/XTS/Mover.TcPOU
FUNCTION_BLOCK Mover
VAR_INPUT
	Enable			: BOOL;				// Request mover enable
	toStart			: BOOL;				// Request mover go to start position
	toNext			: BOOL;				// Request mover go to next station	
	toStop			: BOOL;				// Request mover to stop - meaning the movers will be stop, removed from group, and power will be shutdown to the track via an E-Stop or HMI.Stop	
	toPause			: BOOL;				// Request mover to pause	
	toDisable		: BOOL;				// Request mover to disable power	
	toQueue			: BOOL;				// Request current mover at starting station to join the back of the queue
	toReset			: BOOL;				// Request current mover at starting station to join the back of the queue
END_VAR
VAR_OUTPUT
	Enabled			: BOOL;				// Mover confirmed enabled
	Ready			: BOOL;				// Mover is enabled and ready to accept motion commands
	Busy			: BOOL;				// Mover is processing a command or changing state
	Position		: LREAL;			// Current mover position
	Velocity		: LREAL;			// Current mover velocity                                	
	Error			: UDINT;			// errorID of the active error
	Step			: MoverSequence;	// Mover's step within sequence                                	
	AxisReference	: AXIS_REF;			// Motion link variable. Left as output so the link can be made directly, and accessed by external code
	TargetStation	: USINT;
END_VAR
VAR
	// Motion commands
	fbPower					: MC_Power;
	fbReset					: MC_Reset;
	fbHaltCA				: MC_HaltCA;
	fbMoveAbsCA				: MC_MoveAbsoluteCA;
	fbMoveAbsCABlended		: MC_MoveAbsoluteCA;
	
	MoveCommandVel			: LREAL := 400;
	PosLow					: LREAL;
	PosHigh					: LREAL;
	
END_VAR

(* this function block handles each Mover's axis *)

// feedback



	AxisReference.ReadStatus();

	Enabled		:= NOT AxisReference.Status.Disabled;
	Ready		:= AxisReference.Status.NotMoving AND NOT AxisReference.Status.Error AND NOT AxisReference.Status.Disabled;
	Busy		:= AxisReference.Status.Moving;
	Position	:= AxisReference.NcToPlc.ModuloActPos;
	Velocity	:= AxisReference.NcToPlc.ActVelo;
	Error		:= AxisReference.NcToPlc.ErrorCode;
	
	IF Step = MoverSequence.AtStart AND toQueue THEN
		Step := MoverSequence.MovingToQueue;
		toQueue := FALSE;
	END_IF
	
	

	IF toStop OR toPause THEN
		fbMoveAbsCA.Execute		:= FALSE;
		fbHaltCA.Execute 		:= TRUE;
		fbHaltCA.Deceleration 	:= 1E4;
		IF toStop THEN
			Step := MoverSequence.Stopping;
		ELSIF toPause THEN
			Step := MoverSequence.Pausing;
		END_IF
	END_IF
	
	IF toReset THEN
		Step := MoverSequence.Reset;
		toReset := FALSE;
	END_IF

CASE Step OF
	//-----------------------------------------------------------------------------------------------------------------------
	MoverSequence.Reset:	
	
	fbReset.Execute := TRUE;
	IF fbReset.Busy THEN
		Step := MoverSequence.Resetting;
	END_IF
	
	//-----------------------------------------------------------------------------------------------------------------------
	MoverSequence.Resetting:	
	
	IF fbReset.Done THEN
		fbReset.Execute := FALSE;
		Step := MoverSequence.Waiting;
	END_IF

	//-----------------------------------------------------------------------------------------------------------------------
	MoverSequence.MovingToQueue:	
	
	IF NOT fbMoveAbsCA.Busy AND NOT fbMoveAbsCA.Done THEN			//Add additional condition that the doors are not unlcoked
			fbMoveAbsCA.Execute			:= TRUE;
			fbMoveAbsCA.Position		:= GVL.Station[GVL.startStation].Position+2000;
			fbMoveAbsCA.Velocity		:= MoveCommandVel;										// parameterize
			fbMoveAbsCA.Direction		:= MC_Positive_Direction;						// usually positive
		END_IF
		// check for error
		IF fbMoveAbsCA.Error THEN
			Error				:= fbMoveAbsCA.ErrorId;
			Step				:= MoverSequence.Error;
			fbMoveAbsCA.Execute	:= FALSE;
		END_IF
		// check for move complete THEN proceed to starting station
		IF fbMoveAbsCA.Busy AND Position > 1500.0 AND Position < 6900.0 THEN 		//When mover sits at position 0 the values jump +-0 so an asdditional condition must be used
			fbMoveAbsCABlended.Execute		:= TRUE;
			//bDummy							:= TRUE;
			fbMoveAbsCABlended.Position		:= GVL.Station[GVL.startStation].Position;
			fbMoveAbsCABlended.Velocity		:= MoveCommandVel;
			fbMoveAbsCABlended.BufferMode	:= mcAborting;
			fbMoveAbsCABlended.Direction 	:= MC_Positive_Direction;
			Step							:= MoverSequence.AtQueue;
		END_IF
		
	//-----------------------------------------------------------------------------------------------------------------------
	MoverSequence.AtQueue:	
	
	IF fbMoveAbsCABlended.Busy THEN
		fbMoveAbsCABlended.Execute			:= FALSE;
		fbMoveAbsCA.Execute					:= FALSE;
		Step								:= MoverSequence.MovingToStart;
	END_IF
	
	
//-----------------------------------------------------------------------------------------------------------------------
	MoverSequence.Stopping:	
	
		IF fbHaltCA.Done OR AxisReference.Status.StandStill THEN
			fbHaltCA.Execute 	:= FALSE;
			toStart				:= FALSE;
			toNext				:= FALSE;
			toStop				:= FALSE;
			Step := MoverSequence.Disabling;
			END_IF
			
//-----------------------------------------------------------------------------------------------------------------------
	MoverSequence.Disabling:		//RESULT OF PRESSING STOP
	 // Waiting area 
	 
	 IF toDisable THEN
		Enable						:= FALSE;
		fbPower.Enable				:= FALSE;
		fbPower.Enable_Positive		:= FALSE;
		fbPower.Enable_Negative		:= FALSE;
		fbPower.BufferMode			:= MC_Aborting;
		fbPower.Override			:= 100;
		IF AxisReference.Status.Disabled THEN
			toDisable := FALSE;
			Step := MoverSequence.Off;
		END_IF
	END_IF
			
//-----------------------------------------------------------------------------------------------------------------------
	MoverSequence.Pausing:	
	
	
		IF fbHaltCA.Done THEN
			fbHaltCA.Execute 	:= FALSE;
			toStart				:= FALSE;
			toNext				:= FALSE;
			toPause				:= FALSE;
			Step := MoverSequence.OFF;
			END_IF

//-----------------------------------------------------------------------------------------------------------------------
	MoverSequence.Off:
		// when enable request is true, use MC_Power function block
		IF Enable THEN
			fbPower.Enable_Positive := TRUE;
			fbPower.Enable := TRUE;
		END_IF
		IF Enabled THEN
			Step	:= MoverSequence.Idle;
		END_IF
		
//-----------------------------------------------------------------------------------------------------------------------	
	MoverSequence.Idle:
		// ready and awaiting either toStart or toNext
		IF toStart THEN
			TargetStation		:= GVL.startStation;
			Step				:= MoverSequence.MovingToStart;
		ELSIF toNext THEN
			Step				:= MoverSequence.MovingToStation;
		END_IF
		
//-----------------------------------------------------------------------------------------------------------------------	
	MoverSequence.MovingToStart:
		// move absolute with collision avoidance to start station
		IF NOT fbMoveAbsCA.Busy AND NOT fbMoveAbsCA.Done THEN			//Add additional condition that the doors are not unlcoked
			fbMoveAbsCA.Execute			:= TRUE;
			fbMoveAbsCA.Position		:= GVL.Station[GVL.startStation].Position;
			fbMoveAbsCA.Velocity		:= MoveCommandVel;										// parameterize
			fbMoveAbsCA.Direction		:= MC_Positive_Direction;						// usually positive
		ELSE
			fbMoveAbsCA.Execute			:= FALSE;
		END_IF
		// check for error
		IF fbMoveAbsCA.Error THEN
			Error				:= fbMoveAbsCA.ErrorId;
			Step				:= MoverSequence.Error;
			fbMoveAbsCA.Execute	:= FALSE;
		END_IF
		// check for move complete
		IF fbMoveAbsCA.Done OR (Position > -3 AND Position < 3) THEN
			fbMoveAbsCA.Execute	:= FALSE;
			toStart				:= FALSE;
			Step				:= MoverSequence.AtStart;
		END_IF
		
//-----------------------------------------------------------------------------------------------------------------------	
	MoverSequence.AtStart:
		toStart					:= FALSE;							//Add additional condition that the doors are not unlcoked
		// wait for command to next station
		IF toNext THEN
			IF TargetStation < GVL.NUM_STATIONS THEN
				// next station
				TargetStation	:= TargetStation + 1;
			ELSE
				// at last station, next station is 1
				TargetStation	:= 1;
			END_IF
			Step				:= MoverSequence.MovingToStation;
		END_IF
//-----------------------------------------------------------------------------------------------------------------------	
	MoverSequence.MovingToStation:
		// move absolute with collision avoidance to next station		//Add additional condition that the doors are not unlcoked
		fbMoveAbsCA.Execute			:= TRUE;
				fbMoveAbsCA.Position		:= GVL.Station[TargetStation].Position;
				fbMoveAbsCA.Velocity		:= MoveCommandVel;										// parameterize
				fbMoveAbsCA.Direction		:= MC_Positive_Direction;						// usually positive
		// check for error
		IF fbMoveAbsCA.Error THEN
			Error				:= fbMoveAbsCA.ErrorId;
			Step				:= MoverSequence.Error;
			fbMoveAbsCA.Execute	:= FALSE;
		END_IF
		// check for move complete
		IF fbMoveAbsCA.Done THEN
			fbMoveAbsCA.Execute := FALSE;
			toNext				:= FALSE;
			Step				:= MoverSequence.AtStation;
		END_IF
//-----------------------------------------------------------------------------------------------------------------------	
	MoverSequence.AtStation:
		// wait for command to next station
		IF toNext THEN															//Add additional condition that the doors are not unlcoked
			IF TargetStation < GVL.NUM_STATIONS THEN
				// next station
				TargetStation	:= TargetStation + 1;
			ELSE
				// at last station, next station is 1
				TargetStation	:= 1;
			END_IF
			Step				:= MoverSequence.MovingToStation;
		END_IF
		
		IF toStart THEN
			Step				:= MoverSequence.MovingToStart;
		END_IF
		
END_CASE

	fbPower(Axis := AxisReference);
	fbReset(Axis := AxisReference);
	fbHaltCA(Axis := AxisReference);
	fbMoveAbsCA(Axis := AxisReference);
	fbMoveAbsCABlended(Axis := AxisReference);

END_FUNCTION_BLOCK

// ---- POUs/XTS/Station.TcPOU
FUNCTION_BLOCK Station
VAR_INPUT
	Position		: LREAL;
	bMoveToNext		: BOOL;
	bMoveToStart	: BOOL;
	bMoveToQueue	: BOOL;
END_VAR
VAR_OUTPUT
	CurrentMover	: UDINT;
END_VAR
VAR
	Step			: StationSequence;
	i				: USINT;
	PosLow			: LREAL;
	PosHigh			: LREAL;
END_VAR

(* this function block handles each station *)

PosLow		:= Position - ( GVL.stationTolerance / 2 );
IF PosLow < 0 THEN
	PosLow	:= GVL.TRACK_LENGTH + PosLow;
END_IF
PosHigh		:= Position + ( GVL.stationTolerance / 2 );

CASE Step OF 
	StationSequence.Idle:
		// loop through all movers checking position
		FOR i := 1 TO GVL.NUM_MOVERS DO
			IF GVL.Mover[i].Ready
			AND ( GVL.Mover[i].Step = MoverSequence.AtStart OR GVL.Mover[i].Step = MoverSequence.AtStation )
			AND ABS(GVL.Mover[i].Velocity) < GVL.zeroSpeed THEN
				IF PosLow < PosHigh THEN
					IF GVL.Mover[i].Position > PosLow
					AND GVL.Mover[i].Position < PosHigh THEN
						CurrentMover	:= i;
						Step			:= StationSequence.MoverPresent;
					END_IF
				ELSE
					// station position is close to rollover
					IF GVL.Mover[i].Position > PosLow
					OR GVL.Mover[i].Position < PosHigh THEN
						CurrentMover	:= i;
						Step			:= StationSequence.MoverPresent;
					END_IF
				END_IF
			END_IF
		END_FOR
//-----------------------------------------------------------------------------------------------------------------------	
	StationSequence.MoverPresent:
		// robot tasks complete, discharge mover
		
		IF bMoveToNext THEN									
			Step	:= StationSequence.DischargeMover;
			bMoveToNext := FALSE;
			GVL.Mover[CurrentMover].toNext	:= TRUE;		// request mover move to next station
		END_IF
		
		IF bMoveToStart THEN
			Step	:= StationSequence.DischargeMover;
			bMoveToStart := FALSE;
			GVL.Mover[CurrentMover].toStart	:= TRUE;		// request mover move to Start station
		END_IF
		
		IF bMoveToQueue THEN
			Step	:= StationSequence.DischargeMover;
			bMoveToQueue := FALSE;
			GVL.Mover[CurrentMover].toQueue	:= TRUE;
		END_IF
//-----------------------------------------------------------------------------------------------------------------------		
	StationSequence.DischargeMover:
		// request mover move to next station
		//GVL.Mover[CurrentMover].toNext	:= TRUE;
		// verify mover has left
		IF GVL.Mover[CurrentMover].Busy
			AND GVL.Mover[CurrentMover].Position > (Position + GVL.stationTolerance / 2)
			AND GVL.Mover[CurrentMover].Velocity > GVL.zeroSpeed THEN
			Step	:= StationSequence.Idle;
		END_IF
		
END_CASE

END_FUNCTION_BLOCK

// ---- POUs/XTS/Zone.TcPOU
FUNCTION_BLOCK Zone
VAR_INPUT
END_VAR
VAR_OUTPUT
END_VAR
VAR
END_VAR

//

END_FUNCTION_BLOCK
